TYPE ST_Point :
STRUCT
	x		: LREAL;
	y		: LREAL;
END_STRUCT
END_TYPE

(* stored: Version 1.1.0.1, ProductVersion 3.1.4024.12
   DUT ST_Point: Id {6db15727-68a0-4a6e-8ed9-bfb10a68aa3b} *)
